INTERFACE I_WorkingStation

PROPERTY prTableInPosition : BOOL
GET
END_GET
SET
END_SET
END_PROPERTY

PROPERTY prTableRotationInterlock : BOOL
GET
END_GET
SET
END_SET
END_PROPERTY

PROPERTY prTableRotationRequest : BOOL
GET
END_GET
SET
END_SET
END_PROPERTY

END_INTERFACE

(* stored: Version 1.1.0.1, ProductVersion 3.1.4024.15
   Itf I_WorkingStation: Id {4fc3fe90-c1e8-40cd-ba9f-deea71f0ae85}
   Property prTableInPosition: Id {00874bb4-5315-48b6-982f-041445a42ad3}
   Get Get: Id {0fd855f9-d38b-458c-aa01-78c18a4213c2}
   Set Set: Id {e5e8235a-c12d-4d2a-bcf8-2a22cd4c1480}
   Property prTableRotationInterlock: Id {36e7e1ef-3eca-4e02-9d42-157e2e1fc858}
   Get Get: Id {01bd09b6-9f54-4c2d-b79d-742c5fdb82f3}
   Set Set: Id {dd8d538d-614e-475f-a33a-115fd16c76f1}
   Property prTableRotationRequest: Id {ad483de5-b236-4c2c-82fd-5d0976a0b1c1}
   Get Get: Id {add0ad2f-100e-4e6f-9dce-4eb57c7d81e1}
   Set Set: Id {ec1465b0-7371-47c6-8934-fb1d91ea20f9} *)
